// TwinCAT 3 PLC project Oefeningen2
// ProgramVersion: 3.1.4026.18
// libraries:
//   Tc2_BABasic, * (Beckhoff Automation GmbH)
//   Tc2_Standard, * (Beckhoff Automation GmbH)
//   Tc2_System, * (Beckhoff Automation GmbH)
//   Tc3_Module, * (Beckhoff Automation GmbH)
//   VisuDialogs, * (System)
// project tree:
//   / GlobalTextList.TcGTLO, PlcTask.TcTTO, Visualization Manager.TcVMO (not stored)
//   POUs/ MAIN.TcPOU, prg_DynamischVerschalen.TcPOU, prg_PotentioMeter.TcPOU, prg_Processbewaking3Vaten.TcPOU, prg_TolerantiesEnHysteresis.TcPOU, prg_VerschalenDisplay.TcPOU
//   VISUs/ Visualization_DynamischVerschalen.TcVIS
// (motion and I/O tree: see PLC project oefeningen1)
// real-time tasks:
//   TASK PlcTask: cycle T#10ms, priority 20, ADS port 350
//   TASK PlcTask1: cycle T#10ms, priority 21, ADS port 351
//   TASK PlcTask2: cycle T#10ms, priority 22, ADS port 352
//   TASK PlcTask3: cycle T#10ms, priority 23, ADS port 353
//   TASK PlcTask4: cycle T#10ms, priority 24, ADS port 354

CONFIGURATION Oefeningen2
    RESOURCE PLC ON TwinCAT3
        TASK PlcTask(INTERVAL := T#10ms, PRIORITY := 21);
        PROGRAM MAIN WITH PlcTask : MAIN;
    END_RESOURCE
END_CONFIGURATION

// ---- POUs/MAIN.TcPOU
PROGRAM MAIN
VAR
END_VAR

//prg_PotentioMeter();
prg_DynamischVerschalen();
//prg_TolerantiesEnHysteresis();
//prg_VerschalenDisplay();
//prg_Processbewaking3Vaten();

END_PROGRAM

// ---- POUs/prg_DynamischVerschalen.TcPOU
PROGRAM prg_DynamischVerschalen
VAR
	nPotentioMeter		AT		%I*		:INT;
	
	nPotPower			AT		%Q*		:INT := 32767; //Potentiometer voeden met 5V
	nWaarde				AT		%Q*		:REAL;
	nScaledMax			AT		%Q*		:INT;
END_VAR

//nScaledMax := 10; IN VISU GEKOZEN
nWaarde := INT_TO_REAL(nPotentioMeter) * INT_TO_REAL(nScaledMax) / 32767;

//Andere oplossing:
//nScaledMax := 10;
//nWaarde := INT_TO_REAL(nPotentioMeter) * nScaledMax) / 32767;

END_PROGRAM

// ---- POUs/prg_PotentioMeter.TcPOU
PROGRAM prg_PotentioMeter
VAR
	nPotentioMeter		AT		%I*		:INT;
	
	nPotPower			AT		%Q*		:INT := 32767; //Potentiometer voeden met 5V
	nWaarde				AT		%Q*		:REAL;
END_VAR

nWaarde := INT_TO_REAL(nPotentioMeter)*100 / 32767;

//Ander Oplossing:
//nWaarde:= INT_TO_REAL(nPotentioMeter) /327.67;

END_PROGRAM

// ---- POUs/prg_Processbewaking3Vaten.TcPOU
PROGRAM prg_Processbewaking3Vaten
VAR
	nVatWaarde1, nVatWaarde2, nVatWaarde3		AT		%I*		:INT;
	nVat1, nVat2, nVat3							AT		%Q*		:INT;
END_VAR

nVat1 := nVatWaarde1 * 2000 /32767;
nVat2 := nVatWaarde2 * 3000 /32767;
nVat3 := nVatWaarde3 * 5000 /32767;

//Of misschien beter voor afronding maar onnodig lang:
//nVat1 := REAL_TO_INT(INT_TO_REAL(nVatWaarde1) * 2000 / 32767);
//nVat2 := REAL_TO_INT(INT_TO_REAL(nVatWaarde2) * 3000 / 32767);
//nVat3 := REAL_TO_INT(INT_TO_REAL(nVatWaarde3) * 5000 / 32767);

END_PROGRAM

// ---- POUs/prg_TolerantiesEnHysteresis.TcPOU
PROGRAM prg_TolerantiesEnHysteresis
VAR
	nTemperatuurGevraagd	AT %I* : REAL;   // via visualisatie (180–230)
	nTemperatuurMeting		AT %I* : INT;    // potentiometer

	nPotPower				AT %Q* : INT := 32767;

	GroeneLed				AT %Q* : BOOL;
	RodeLed					AT %Q* : BOOL;

	nGemeten				: REAL;
END_VAR

nGemeten := INT_TO_REAL(nTemperatuurMeting) * 250 / 32767;

IF nGemeten < nTemperatuurGevraagd * 0.9 THEN
	RodeLed := TRUE;  GroeneLed := FALSE;
ELSIF nGemeten > nTemperatuurGevraagd * 1.1 THEN
	GroeneLed := TRUE;  RodeLed := FALSE;
END_IF

END_PROGRAM

// ---- POUs/prg_VerschalenDisplay.TcPOU
PROGRAM prg_VerschalenDisplay
VAR
	nPotentioMeter		AT		%I*		:INT;
	
	nPotPower			AT		%Q*		:INT := 32767; //Potentiometer voeden met 5V
	nWaarde				AT		%Q*		:INT;
END_VAR

nWaarde := nPotentioMeter * 1000 / 32767;

//Misschien zelfs beter maar onnodig moeilijke oplossing:
//	nWaarde := REAL_TO_INT(INT_TO_REAL(nPotentioMeter) * 1000 / 32767);

END_PROGRAM

// ---- GlobalTextList.TcGTLO
TEXTLIST GlobalTextList
  943 = 'De max waarde is %d'
  201 = 'De max waarde waarde: %d'
  27 = 'Verschaalde waarde: %d'
END_TEXTLIST

// ---- VISUs/Visualization_DynamischVerschalen.TcVIS
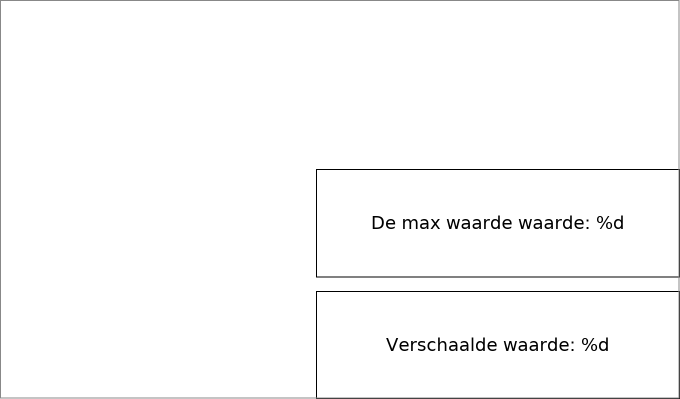
VISUALIZATION Visualization_DynamischVerschalen  // 680x399
    Rectangle (316,291 364x108), "Verschaalde waarde: %d", text variable: prg_DynamischVerschalen.nWaarde
    Rectangle (316,169 364x108), "De max waarde waarde: %d", text variable: prg_DynamischVerschalen.nScaledMax
        OnMouseDown: write the text variable via Default
END_VISUALIZATION
